// TwinCAT 3 PLC project TcoMitsubishiRoboticsTests
// Title: TcoMitsubishiRoboticsTests
// Company: Vortex.Library
// Author: TcOpenGroup
// ProjectVersion: 0.6.0.913
// ProgramVersion: 3.1.4024.12
// libraries:
//   Tc2_EtherCAT, * (Beckhoff Automation GmbH)
//   Tc2_MC2, * (Beckhoff Automation GmbH)
//   Tc2_Standard, * (Beckhoff Automation GmbH)
//   Tc2_System, * (Beckhoff Automation GmbH)
//   Tc3_Module, * (Beckhoff Automation GmbH)
//   TcoAbstractions, 0.6.0.913 (Vortex.Library)
//   TcoCore, 0.6.0.913 (Vortex.Library)
//   TcoIo, 0.6.0.913 (Vortex.Library)
//   TcoMitsubishiRobotics, 0.6.0.913 (Vortex.Library)
//   TcoUtilities, 0.6.0.913 (Vortex.Library)
// project tree:
//   GVLs/ GVL.TcGVL
//   / PlcTask1.TcTTO
//   POUs/ MAIN.TcPOU
//   Tests/TcoContext/ SequenceTask.TcPOU, WpfContext.TcPOU
//   Tests/TcoMitsubishiRobotics/ eTcoMitsubishiRoboticsSimpleTests.TcDUT, TcoTestContext.TcPOU, TcoMitsubishiRoboticsTest.TcPOU
// (motion and I/O tree: see PLC project tcomitsubishirobotics)
// real-time tasks:
//   TASK PlcTask: cycle T#10ms, priority 20, ADS port 350
//   TASK PlcTask1: cycle T#10ms, priority 1, ADS port 351
//   TASK PN: cycle T#8ms, priority 2, ADS port 301
// variable links:
//   TcoMitsubishiRoboticsTests/TcoMitsubishiRoboticsTests Instance <-> Device 3 (EL6631)/robot
//     PlcTask1 Inputs/GVL.Robot1.In.Inputs[{0..63}] <-> API/Term 10 (In/Out  64 byte)/Subterm 20 (In/Out  64 byte)/Inputs/Input[{0..63}]  (64 links)
//     PlcTask1 Inputs/GVL.Robot1.PnIoBoxDiag <-> Inputs/PnIoBoxDiag
//     PlcTask1 Inputs/GVL.Robot1.PnIoBoxState <-> Inputs/PnIoBoxState
//     PlcTask1 Outputs/GVL.Robot1.Out.Outputs[{0..63}] <-> API/Term 10 (In/Out  64 byte)/Subterm 20 (In/Out  64 byte)/Outputs/Output[{0..63}]  (64 links)

CONFIGURATION TcoMitsubishiRoboticsTests
    RESOURCE PLC ON TwinCAT3
        TASK PlcTask1(INTERVAL := T#10ms, PRIORITY := 1);
        PROGRAM MAIN WITH PlcTask1 : MAIN;
    END_RESOURCE
END_CONFIGURATION

// ---- Tests/TcoMitsubishiRobotics/eTcoMitsubishiRoboticsSimpleTests.TcDUT
{attribute 'qualified_only'}
{attribute 'strict'}
TYPE eTcoMitsubishiRoboticsSimpleTests :
(
    Restore := 1,
    CleanUp,
    Message,
    PowerDisable,
    PowerEnable,
    Reset,
    MoveRelativePositiveWithDisabledPositiveDirection,
    MoveRelativePositiveWithEnabledPositiveDirection,
    MoveRelativeNegativeWithDisabledNegativeDirection,
    MoveRelativeNegativeWithEnabledNegativeDirection,
    HommingDirect,
    MoveVelocityPositiveWithDisabledPositiveDirection,
    MoveVelocityPositiveWithEnabledPositiveDirection,
    Stop,
    MoveVelocityNegativeWithDisabledNegativeDirection,
    MoveVelocityNegativeWithEnabledNegativeDirection,
    MoveAbsoluteDisabled,
    MoveAbsoluteDisabledPositiveDirection,
    MoveAbsoluteEnabledPositiveDirection,
    MoveAbsoluteDisabledNegativeDirection,
    MoveAbsoluteEnabledNegativeDirection,
    Last
);
END_TYPE

// ---- GVLs/GVL.TcGVL
{attribute 'qualified_only'}
VAR_GLOBAL
    Robot1 : TcoMitsubishiRobotics.TcoCr800_IO_v_1_x_x;
END_VAR

// ---- POUs/MAIN.TcPOU
PROGRAM MAIN
VAR
    _tcoTestContext : TcoTestContext;
    _wpfContext : WpfContext;
    _wpfContextCall : BOOL := FALSE;
END_VAR

_tcoTestContext.ProbeRun();

IF _wpfContextCall THEN
    _wpfContext.Run();
END_IF

END_PROGRAM

// ---- Tests/TcoMitsubishiRobotics/TcoTestContext.TcPOU
FUNCTION_BLOCK TcoTestContext EXTENDS TcoCore._internals_TcoContext
VAR
    _sut : TcoMitsubishiRoboticsTest(THIS^);
    _callMyPlcInstance : BOOL := FALSE;
    _enable : BOOL;
    _enablePositive : BOOL;
    _enableNegative : BOOL;
    _calibrationCam : BOOL;
    _position : LREAL;
    _velocity : LREAL;
    _acceleration : LREAL;
    _deceleration : LREAL;
    _jerk : LREAL;
    _inString : STRING;
    _done : BOOL;
    _arranged : BOOL;
    _axisReferenceType : INT;
END_VAR

METHOD PROTECTED Main
//_sut(inEnable := _enable,
//    inEnablePositive := _enablePositive,
//    inEnableNegative := _enableNegative,
//    inCalibrationCam := _calibrationCam,
//    inoAxisRef := GVL.Axis1);
//
//CASE _testId OF
//    eTcoDriveSimpleTests.Restore:
//        _sut.Restore();
//    eTcoDriveSimpleTests.CleanUp:
//        _sut._messenger.Clear();
//    {region "T003_Message"}
//    eTcoDriveSimpleTests.Message:
//        _sut.Messenger.Error(_inString);
//        _done := _plcCycleCounter > 1;
//        ProbeDoneWhen(_done);
//    {endregion}
//    {region "T004_PowerDisable"}
//    eTcoDriveSimpleTests.PowerDisable:
//        _enable := FALSE;
//        _done := _sut._axisStatus.Disabled; // OR _plcCycleCounter > 1;
//        ProbeDoneWhen(_done);
//    {endregion}
//    {region "T005_PowerEnable"}
//    eTcoDriveSimpleTests.PowerEnable:
//        _enable := TRUE;
//        _done := _sut._axisStatus.Operational; // OR _plcCycleCounter > 15;
//        ProbeDoneWhen(_done);
//    {endregion}
//    {region "T006_Reset"}
//    eTcoDriveSimpleTests.Reset:
//        IF NOT _arranged THEN
//            _sut.MoveRelative(inDistance := 500,
//                inVelocity := 50000000,
//                inAcceleration := -1,
//                inDeceleration := -1,
//                inJerk := -1);
//
//            IF _sut._axisStatus.Error THEN
//                _arranged := true;
//            END_IF
//
//            RETURN;
//        END_IF
//
//        _sut.Reset();
//        _done := _sut.ResetTask.Done OR _sut.ResetTask.Error; // OR _plcCycleCounter > 1;
//        ProbeDoneWhen(_done);
//    {endregion}
//    {region "T007_MoveRelativePositiveWithDisabledPositiveDirection"}
//    eTcoDriveSimpleTests.MoveRelativePositiveWithDisabledPositiveDirection:
//        IF NOT _arranged THEN
//            _enable := TRUE;
//            _enablePositive := FALSE;
//            _enableNegative := FALSE;
//
//            IF _sut._axisStatus.Operational THEN
//                _arranged := TRUE;
//            END_IF
//
//            RETURN;
//        END_IF;
//
//        _sut.MoveRelative(inDistance := _position,
//            inVelocity := _velocity,
//            inAcceleration := _acceleration,
//            inDeceleration := _deceleration,
//            inJerk := _jerk);
//
//        _done := _sut.MoveRelativeTask.Done OR _sut.MoveRelativeTask.Error; // OR _sut._axisStatus.Error;// OR _plcCycleCounter > 5;
//        ProbeDoneWhen(_done);
//    {endregion}
//    {region "T008_MoveRelativePositiveWithEnabledPositiveDirection"}
//    eTcoDriveSimpleTests.MoveRelativePositiveWithEnabledPositiveDirection:
//        IF NOT _arranged THEN
//            _enable := TRUE;
//            _enablePositive := TRUE;
//            _enableNegative := FALSE;
//
//            IF _sut._axisStatus.Operational THEN
//                _arranged := TRUE;
//            END_IF
//
//            RETURN;
//        END_IF;
//
//        _sut.MoveRelative(inDistance := _position,
//            inVelocity := _velocity,
//            inAcceleration := _acceleration,
//            inDeceleration := _deceleration,
//            inJerk := _jerk);
//
//        _done := _sut.MoveRelativeTask.Done OR _sut.MoveRelativeTask.Error; // OR  _plcCycleCounter > 1000;
//        ProbeDoneWhen(_done);
//    {endregion}
//    {region "T009_MoveRelativeNegativeWithDisabledNegativeDirection"}
//    eTcoDriveSimpleTests.MoveRelativeNegativeWithDisabledNegativeDirection:
//        IF NOT _arranged THEN
//            _enable := TRUE;
//            _enablePositive := FALSE;
//            _enableNegative := FALSE;
//
//            IF _sut._axisStatus.Operational THEN
//                _arranged := TRUE;
//            END_IF
//
//            RETURN;
//        END_IF;
//
//        _sut.MoveRelative(inDistance := _position,
//            inVelocity := _velocity,
//            inAcceleration := _acceleration,
//            inDeceleration := _deceleration,
//            inJerk := _jerk);
//
//        _done := _sut.MoveRelativeTask.Done OR _sut.MoveRelativeTask.Error; // OR _sut._axisStatus.Error;// OR _plcCycleCounter > 5;
//        ProbeDoneWhen(_done);
//    {endregion}
//    {region "T010_MoveRelativeNegativeWithEnabledNegativeDirection"}
//    eTcoDriveSimpleTests.MoveRelativeNegativeWithEnabledNegativeDirection:
//        IF NOT _arranged THEN
//            _enable := TRUE;
//            _enablePositive := TRUE;
//            _enableNegative := TRUE;
//
//            IF _sut._axisStatus.Operational THEN
//                _arranged := TRUE;
//            END_IF
//
//            RETURN;
//        END_IF;
//
//        _sut.MoveRelative(inDistance := _position,
//            inVelocity := _velocity,
//            inAcceleration := _acceleration,
//            inDeceleration := _deceleration,
//            inJerk := _jerk);
//
//        _done := _sut.MoveRelativeTask.Done OR _sut.MoveRelativeTask.Error; // OR  _plcCycleCounter > 1000;
//        ProbeDoneWhen(_done);
//    {endregion}
//    {region "T011_HommingDirect"}
//    eTcoDriveSimpleTests.HommingDirect:
//        IF NOT _arranged THEN
//            _enable := TRUE;
//            _enablePositive := FALSE;
//            _enableNegative := TRUE;
//
//            IF _sut._axisStatus.Operational THEN
//                _arranged := TRUE;
//            END_IF
//
//            RETURN;
//        END_IF;
//
//        _sut.Home(inPosition := _position,
//            inHomingMode := TcoDrivesBeckhoff.eHomingMode.MC_Direct,
//            inClearPositionLag := FALSE,
//            inSearchDirection := TcoDrivesBeckhoff.eDirection.MC_Undefined_Direction,
//            inSearchVelocity := _velocity,
//            inSyncDirection := TcoDrivesBeckhoff.eDirection.MC_Undefined_Direction,
//            inSyncVelocity := _velocity,
//            inReferenceMode := TcoDrivesBeckhoff.eEncoderReferenceMode.ENCODERREFERENCEMODE_DEFAULT);
//
//        _done := _sut.HomeTask.Done OR _sut.HomeTask.Error; //OR _plcCycleCounter > 1000;
//        ProbeDoneWhen(_done);
//    {endregion}
//    {region "T012_MoveVelocityPositiveWithDisabledPositiveDirection"}
//    eTcoDriveSimpleTests.MoveVelocityPositiveWithDisabledPositiveDirection:
//        IF NOT _arranged THEN
//            _enable := TRUE;
//            _enablePositive := FALSE;
//            _enableNegative := FALSE;
//
//            IF _sut._axisStatus.Operational THEN
//                _arranged := TRUE;
//            END_IF
//
//            RETURN;
//        END_IF;
//
//        _sut.MoveVelocity(inVelocity := _velocity,
//            inAcceleration := _acceleration,
//            inDeceleration := _deceleration,
//            inJerk := _jerk,
//            inDirection := TcoDrivesBeckhoff.eDirection.MC_Positive_Direction);
//
//        _done := _sut.MoveVelocityTask.Done OR _sut.MoveVelocityTask.Error; // OR  _sut._axisStatus.Error;// OR _plcCycleCounter > 5;
//        ProbeDoneWhen(_done);
//    {endregion}
//    {region "T013_MoveVelocityPositiveWithEnabledPositiveDirection"}
//    eTcoDriveSimpleTests.MoveVelocityPositiveWithEnabledPositiveDirection:
//        IF NOT _arranged THEN
//            _enable := TRUE;
//            _enablePositive := TRUE;
//            _enableNegative := FALSE;
//
//            IF _sut._axisStatus.Operational THEN
//                _arranged := TRUE;
//            END_IF
//
//            RETURN;
//        END_IF;
//
//        _sut.MoveVelocity(inVelocity := _velocity,
//            inAcceleration := _acceleration,
//            inDeceleration := _deceleration,
//            inJerk := _jerk,
//            inDirection := TcoDrivesBeckhoff.eDirection.MC_Positive_Direction);
//
//        _done := _sut.MoveVelocityTask.Done OR _sut.MoveVelocityTask.Error; // OR  _plcCycleCounter > 1000;
//        ProbeDoneWhen(_done);
//    {endregion}
//    {region "T014_Stop"}
//    eTcoDriveSimpleTests.Stop:
//        IF NOT _arranged THEN
//            _enable := TRUE;
//            _enablePositive := TRUE;
//            _enableNegative := TRUE;
//
//            IF _sut._axisStatus.Operational THEN
//                _arranged := TRUE;
//            END_IF
//
//            RETURN;
//        END_IF;
//
//        _sut.Stop(inDeceleration := _deceleration, inJerk := _jerk);
//        _done := _sut.StopTask.Done OR _sut.StopTask.Error; // OR  _plcCycleCounter > 1000;
//        ProbeDoneWhen(_done);
//    {endregion}
//    {region "T015_MoveVelocityNegativeWithDisabledNegativeDirection"}
//    eTcoDriveSimpleTests.MoveVelocityNegativeWithDisabledNegativeDirection:
//        IF NOT _arranged THEN
//            _enable := TRUE;
//            _enablePositive := FALSE;
//            _enableNegative := FALSE;
//
//            IF _sut._axisStatus.Operational THEN
//                _arranged := TRUE;
//            END_IF
//
//            RETURN;
//        END_IF;
//
//        _sut.MoveVelocity(inVelocity := _velocity,
//            inAcceleration := _acceleration,
//            inDeceleration := _deceleration,
//            inJerk := _jerk,
//            inDirection := TcoDrivesBeckhoff.eDirection.MC_Negative_Direction);
//
//        _done := _sut.MoveVelocityTask.Done OR _sut.MoveVelocityTask.Error; // OR  _sut._axisStatus.Error;// OR _plcCycleCounter > 5;
//        ProbeDoneWhen(_done);
//    {endregion}
//    {region "T016_MoveVelocityNegativeWithEnabledNegativeDirection"}
//    eTcoDriveSimpleTests.MoveVelocityNegativeWithEnabledNegativeDirection:
//        IF NOT _arranged THEN
//            _enable := TRUE;
//            _enablePositive := FALSE;
//            _enableNegative := TRUE;
//
//            IF _sut._axisStatus.Operational THEN
//                _arranged := TRUE;
//            END_IF
//
//            RETURN;
//        END_IF;
//
//        _sut.MoveVelocity(inVelocity := _velocity,
//            inAcceleration := _acceleration,
//            inDeceleration := _deceleration,
//            inJerk := _jerk,
//            inDirection := TcoDrivesBeckhoff.eDirection.MC_Negative_Direction);
//
//        _done := _sut.MoveVelocityTask.Done OR _sut.MoveVelocityTask.Error; // OR  _plcCycleCounter > 1000;
//        ProbeDoneWhen(_done);
//    {endregion}
//    {region "T017_MoveAbsoluteDisabled"}
//    eTcoDriveSimpleTests.MoveAbsoluteDisabled:
//        IF NOT _arranged THEN
//            _enable := FALSE;
//            _enablePositive := FALSE;
//            _enableNegative := FALSE;
//            _arranged := TRUE;
//            RETURN;
//        END_IF;
//
//        _sut.MoveAbsolute(inPosition := _position,
//            inVelocity := _velocity,
//            inAcceleration := _acceleration,
//            inDeceleration := _deceleration,
//            inJerk := _jerk);
//
//        _done := _sut.MoveAbsoluteTask.Done OR _sut.MoveAbsoluteTask.Error OR _plcCycleCounter > 10;
//        ProbeDoneWhen(_done);
//	{endregion}
//    {region "T018_MoveAbsoluteDisabledPositiveDirection"}
//    eTcoDriveSimpleTests.MoveAbsoluteDisabledPositiveDirection:
//        IF NOT _arranged THEN
//            _enable := TRUE;
//            _enablePositive := FALSE;
//            _enableNegative := TRUE;
//            _arranged := TRUE;
//            RETURN;
//        END_IF;
//
//        _sut.MoveAbsolute(inPosition := _position,
//            inVelocity := _velocity,
//            inAcceleration := _acceleration,
//            inDeceleration := _deceleration,
//            inJerk := _jerk);
//
//        _done := _sut.MoveAbsoluteTask.Done OR _sut.MoveAbsoluteTask.Error; // OR _sut._axisStatus.Error;// OR _plcCycleCounter > 5;
//        ProbeDoneWhen(_done);
//	{endregion}
//    {region "T019_MoveAbsoluteEnabledPositiveDirection"}
//    eTcoDriveSimpleTests.MoveAbsoluteEnabledPositiveDirection:
//        IF NOT _arranged THEN
//            _enable := TRUE;
//            _enablePositive := TRUE;
//            _enableNegative := FALSE;
//            _arranged := TRUE;
//            RETURN;
//        END_IF;
//
//        _sut.MoveAbsolute(inPosition := _position,
//            inVelocity := _velocity,
//            inAcceleration := _acceleration,
//            inDeceleration := _deceleration,
//            inJerk := _jerk);
//
//        _done := _sut.MoveAbsoluteTask.Done OR _sut.MoveAbsoluteTask.Error; // OR _sut._axisStatus.Error;// OR _plcCycleCounter > 5;
//        ProbeDoneWhen(_done);
//	{endregion}
//    {region "T020_MoveAbsoluteDisabledNegativeDirection"}
//    eTcoDriveSimpleTests.MoveAbsoluteDisabledNegativeDirection:
//        IF NOT _arranged THEN
//            _enable := TRUE;
//            _enablePositive := FALSE;
//            _enableNegative := FALSE;
//            _arranged := TRUE;
//            RETURN;
//        END_IF;
//
//        _sut.MoveAbsolute(inPosition := _position,
//            inVelocity := _velocity,
//            inAcceleration := _acceleration,
//            inDeceleration := _deceleration,
//            inJerk := _jerk);
//
//        _done := _sut.MoveAbsoluteTask.Done OR _sut.MoveAbsoluteTask.Error; // OR _sut._axisStatus.Error;// OR _plcCycleCounter > 5;
//        ProbeDoneWhen(_done);
//	{endregion}
//    {region "T021_MoveAbsoluteEnabledNegativeDirection"}
//    eTcoDriveSimpleTests.MoveAbsoluteEnabledNegativeDirection:
//        IF NOT _arranged THEN
//            _enable := TRUE;
//            _enablePositive := FALSE;
//            _enableNegative := TRUE;
//            _arranged := TRUE;
//            RETURN;
//        END_IF;
//
//        _sut.MoveAbsolute(inPosition := _position,
//            inVelocity := _velocity,
//            inAcceleration := _acceleration,
//            inDeceleration := _deceleration,
//            inJerk := _jerk);
//
//        _done := _sut.MoveAbsoluteTask.Done OR _sut.MoveAbsoluteTask.Error; // OR _sut._axisStatus.Error;// OR _plcCycleCounter > 5;
//        ProbeDoneWhen(_done);
//	{endregion}
//END_CASE
END_METHOD

END_FUNCTION_BLOCK

// ---- Tests/TcoMitsubishiRobotics/TcoMitsubishiRoboticsTest.TcPOU
FUNCTION_BLOCK TcoMitsubishiRoboticsTest EXTENDS TcoMitsubishiRobotics.TcoCr800_v_1_x_x
VAR
    _serviceModeCount : ULINT;
    _serviceModeOverride : LREAL;
END_VAR
VAR
END_VAR

//SUPER^(	inEnable 			:=	inEnable,
//		inEnablePositive	:=	inEnablePositive,
//		inEnableNegative	:=	inEnableNegative,
//		inCalibrationCam	:=	inCalibrationCam,
//		inoAxisRef			:=	inoAxisRef);
//

END_FUNCTION_BLOCK

// ---- Tests/TcoContext/WpfContext.TcPOU
FUNCTION_BLOCK WpfContext EXTENDS TcoCore.TcoContext
VAR
    _serviceModeActive : BOOL;
    {attribute addProperty Name "<#Mitsubichi Cr800#>"}
    _robot1 : TcoMitsubishiRobotics.TcoCr800_v_1_x_x(THIS^);
    _sequence1 : TcoCore.TcoSequence(THIS^, eRestoreMode.None);
    _observer : TcoCore.TcoSequencerObserver(THIS^);
    {attribute addProperty Name "Start sequence"}
    _sequence1Task : SequenceTask(THIS^);
    _dialog : TcoCore.TcoDialog(THIS^);
    _sequence2 : TcoCore.TcoSequence(THIS^, eRestoreMode.None);
    _observer2 : TcoCore.TcoSequencerObserver(THIS^);
    {attribute addProperty Name "Start sequence"}
    _sequence2Task : SequenceTask(THIS^);
    _enable : BOOL;
END_VAR

(*~
    <docu>
        <summary>
            Main method of the TcoContext. This is the entry point of any control logic that belongs to this context.
            The call of this method is ensured by calling the <c>InstanceName.Run()</c> method, and it must not be called explicitly.
            This method is abstract, and it must be overridden in derived block.
        </summary>
    </docu>
~*)
METHOD PROTECTED Main
IF _serviceModeActive THEN
    _robot1.Service();
END_IF

_robot1(inPnIoBoxDiag := GVL.Robot1.PnIoBoxDiag, inPnIoBoxState := gvl.Robot1.PnIoBoxState, inoData := GVL.Robot1);
_sequence1Task.Enabled := NOT _sequence2Task.Busy;
_sequence1Task(Sequence := _sequence1);

IF (_sequence1Task.Execute()) THEN
    Sequence1();
END_IF;
END_METHOD

METHOD Sequence1
VAR
    seq : REFERENCE TO TcoCore.TcoSequence;
    answer : TcoCore.eDialogAnswer;
    done : BOOL;
    _jerk : LREAL;
    _deceleration : LREAL;
    _acceleration : LREAL;
    _velocity : LREAL;
    ProbeDoneWhen : INT;
    _param : TcoRoboticsMovementsParams;
END_VAR
VAR_INST
    _maxAllowedAttempts : INT;
    _noOfAttmets : INT;
END_VAR
seq REF= _sequence1;
seq.Open();
seq.Observer := _observer;

IF (seq.Step(inStepID := 0, inEnabled := TRUE, inStepDescription := 'READY TO START')) THEN
    //--------------------------------------------------------
    _param.GlobalSpeed := 100;
    _noOfAttmets := 0;

    answer := _dialog.Show()
        .WithType(eDialogType.Question)
        .WithCaption('Ready to go?')
        .WithText('Do you really want to start movements? Do we go ahead?')
        .WithYesNo().Answer;

    //
    IF (answer = TcoCore.eDialogAnswer.Yes) THEN
        seq.CompleteStep();
    ELSIF (answer = TcoCore.eDialogAnswer.No) THEN
        _sequence1Task.Restore();
    END_IF;
    //--------------------------------------------------------
END_IF;

IF (seq.Step(inStepID := 10, inEnabled := TRUE, inStepDescription := 'RESTORE')) THEN
    //--------------------------------------------------------
    _robot1.Restore();
    seq.CompleteStep();
    //--------------------------------------------------------
END_IF;

IF (seq.Step(inStepID := 11, inEnabled := TRUE, inStepDescription := 'STOP MOVEMENTS AND PROGRAM')) THEN
    //--------------------------------------------------------
    IF _robot1.StopMovementsAndProgram(inStopType := eTcoRoboticsStopType.Soft).Done THEN
        seq.CompleteStep();
    END_IF

    //--------------------------------------------------------
END_IF;

IF (seq.Step(inStepID := 12, inEnabled := TRUE, inStepDescription := 'START AT MAIN')) THEN
    //--------------------------------------------------------
    IF _robot1.StartAtMain().Done THEN
        seq.CompleteStep();
    END_IF;
    //--------------------------------------------------------
END_IF;

IF (seq.Step(inStepID := 13, inEnabled := TRUE, inStepDescription := 'START MOTORS AND PROGRAM')) THEN
    //--------------------------------------------------------
    IF _robot1.StartMotorsAndProgram().Done THEN
        seq.CompleteStep();
    END_IF;
    //--------------------------------------------------------
END_IF;

IF (seq.Step(inStepID := 14, inEnabled := TRUE, inStepDescription := 'START MOVEMENTS')) THEN
    //--------------------------------------------------------
    _maxAllowedAttempts := 10;
    seq.CompleteStep();
    //--------------------------------------------------------
END_IF;

IF (seq.Step(inStepID := 15, inEnabled := TRUE, inStepDescription := 'START MOVEMENTS')) THEN
    //--------------------------------------------------------
    _param.ActionNo := 100;

    IF _robot1.StartMovements(inData := _param).Done THEN
        seq.CompleteStep();
        _robot1.Restore();
    END_IF
    //--------------------------------------------------------
END_IF;

IF (seq.Step(inStepID := 16, inEnabled := TRUE, inStepDescription := 'START ANOTHER MOVE MOVEMENTS')) THEN
    //--------------------------------------------------------
    _param.ActionNo := 1;
    _param.GlobalSpeed := 90;

    IF _robot1.StartMovements(inData := _param).Done THEN
        IF _noOfAttmets < _maxAllowedAttempts THEN
            _noOfAttmets := _noOfAttmets + 1;
            seq.RequestStep(14);
            _robot1.Restore();
        ELSE
            seq.CompleteStep();
        end_if;
    END_IF
    //--------------------------------------------------------
END_IF;

//
IF (seq.Step(inStepID := 500, inEnabled := TRUE, inStepDescription := 'EXAMPLE OF MOVMENT ABORTED')) THEN
    //    --------------------------------------------------------
    answer := _dialog.Show()
        .WithType(eDialogType.Question)
        .WithCaption('Abort movement?')
        .WithText('Do you  want to start movements and abort it?')
        .WithYesNo().Answer;

    IF (answer = TcoCore.eDialogAnswer.Yes) THEN
        seq.CompleteStep();
    ELSIF (answer = TcoCore.eDialogAnswer.No) THEN
        _sequence1Task.Restore();
    END_IF;
    //    --------------------------------------------------------
END_IF;

IF (seq.Step(inStepID := 525, inEnabled := TRUE, inStepDescription := 'STOP MOVEMENT  EXAMPLE')) THEN
    //    --------------------------------------------------------
    answer :=
        _dialog.Show().WithType(eDialogType.Question).WithCaption('Movement running').WithText('Do you  want to abort movement?').WithYesNo().Answer;

    IF (answer = TcoCore.eDialogAnswer.Yes) THEN
        _robot1.StopMovements(inStopType := TcoAbstractions.eTcoRoboticsStopType.Quick);
        seq.CompleteStep();
    ELSIF (answer = TcoCore.eDialogAnswer.No) THEN
        _sequence1Task.Restore();
    END_IF;

    _param.ActionNo := 100;
    _param.GlobalSpeed := 20;

    IF _robot1.StartMovements(inData := _param).Done THEN
        seq.CompleteStep();
    END_IF
    //    --------------------------------------------------------
END_IF;

IF (seq.Step(inStepID := 600, inEnabled := TRUE, inStepDescription := 'ASKING FOR RESTORING')) THEN
    //    --------------------------------------------------------
    answer := _dialog.Show()
        .WithType(eDialogType.Question)
        .WithCaption('Question?')
        .WithText('Do you want to restore TcoIrc5 component?')
        .WithYesNo().Answer;

    IF (answer = TcoCore.eDialogAnswer.Yes) THEN
        _robot1.Restore();
        seq.CompleteStep();
    ELSIF (answer = TcoCore.eDialogAnswer.No) THEN
        _sequence1Task.Restore();
    END_IF;
    //    --------------------------------------------------------
END_IF;

IF (seq.Step(inStepID := seq.RESTORE_STEP_ID, inEnabled := TRUE, inStepDescription := 'RETURN TO THE START OF THE SEQUENCE')) THEN
    //--------------------------------------------------------
    seq.CompleteSequence();
    //--------------------------------------------------------
END_IF;

seq.Close();
END_METHOD

END_FUNCTION_BLOCK

// ---- Tests/TcoContext/SequenceTask.TcPOU
FUNCTION_BLOCK SequenceTask EXTENDS TcoCore.TcoTask
VAR_INPUT
    Sequence : TcoCore.ITcoSequencer;
END_VAR

(*~
    <docu>
        <summary>
            Restores this instance to the Ready state. Can be called explicitly or from within one of the restore mechanisms.
            <para>
                See also <see cref="PlcDocu.TcoCore.TcoTask.AutoRestorable()"/>
            </para>
        </summary>
    </docu>
~*)
METHOD Restore : ITcoRestorable
SUPER^.Restore();
THIS^.Sequence.Restore();
END_METHOD

END_FUNCTION_BLOCK
